PROGRAM MBUS_WZaehler (* hier wird die Klemme, an welche der M-Bus mit den Zählern angeschlossen ist, alle 10ms aufgerufen *)
VAR
	Komm_Klemme_WZaehler		: FB_MBUSKL6781;
	WMZ331_Brennwerttherme				: FB_MBUS_General_Ext;	(*1*)
	WMZ321_BHKW_1						: FB_MBUS_General_Ext;	(*3*)
	WMZ322_BHKW_2						: FB_MBUS_General_Ext;	(*4*)
	WMZ251_Druckluftkompressor			: FB_MBUS_General_Ext;	(*5*)
	WMZ215_PWT_1						: FB_MBUS_General_Ext;	(*6*)
	WMZ261_Ofenkuehlung_Dichtungen		: FB_MBUS_General_Ext;	(*7*)
	WMZ361_Abwaerme_Ofen_Abgasfackel	: FB_MBUS_General_Ext;	(*8*)
	adrBrennwerttherme				: ST_MBus_SecAdr := (udiIdNumber:=16#00474907);
	adrBHKW_1						: ST_MBus_SecAdr := (udiIdNumber:=16#00470996);
	adrBHKW_2						: ST_MBus_SecAdr := (udiIdNumber:=16#00474904);
	adrDruckluftkompressor			: ST_MBus_SecAdr := (udiIdNumber:=16#00552639);
	adrPWT_1						: ST_MBus_SecAdr := (udiIdNumber:=16#00455395);
	adrOfenkuehlung_Dichtungen		: ST_MBus_SecAdr := (udiIdNumber:=16#00482160);
	adrAbwaerme_Ofen_Abgasfackel	: ST_MBus_SecAdr := (udiIdNumber:=16#00482192);

	fbcatch : 	Error_Catch;
	fbcatch2 : 	Error_Catch;
END_VAR

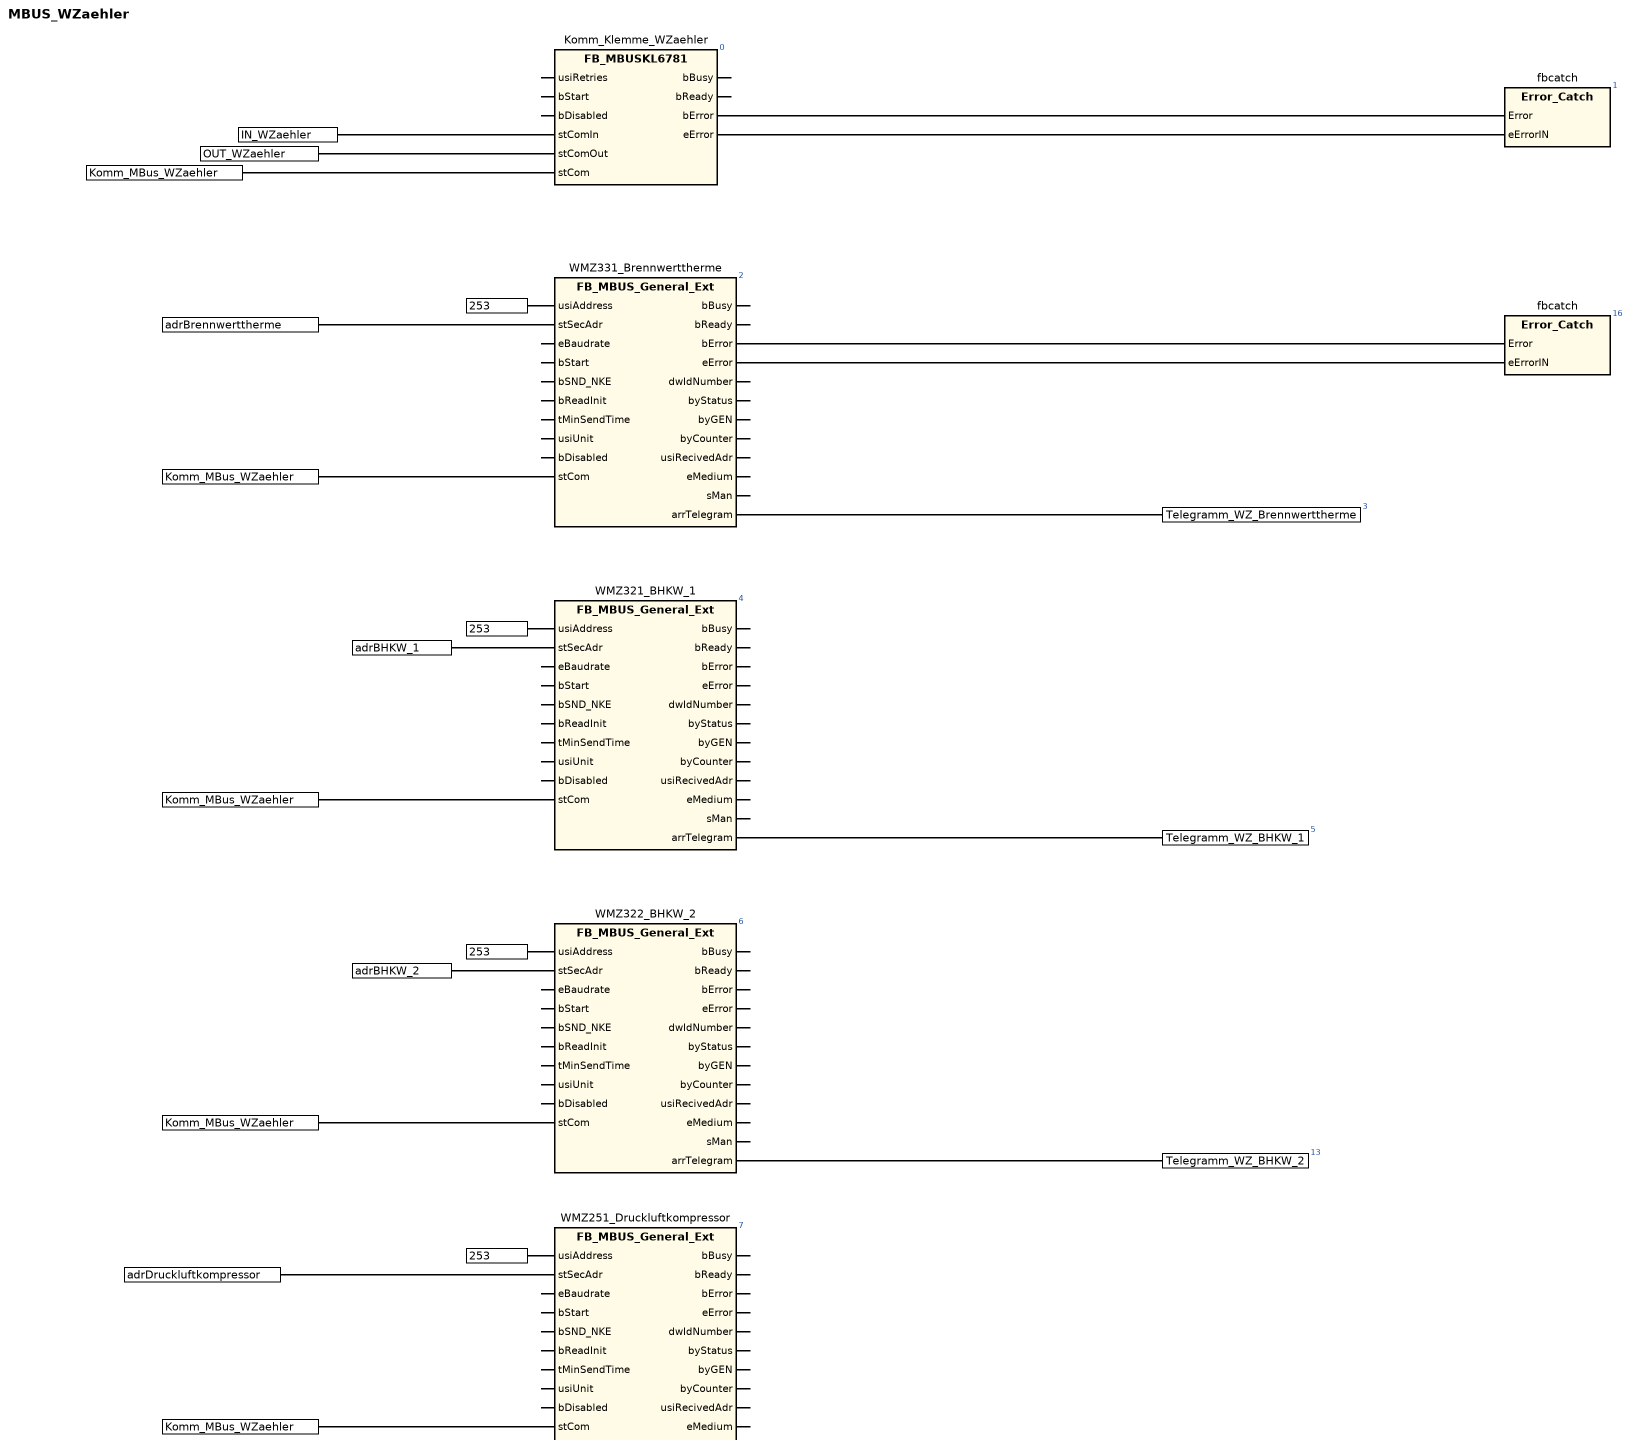
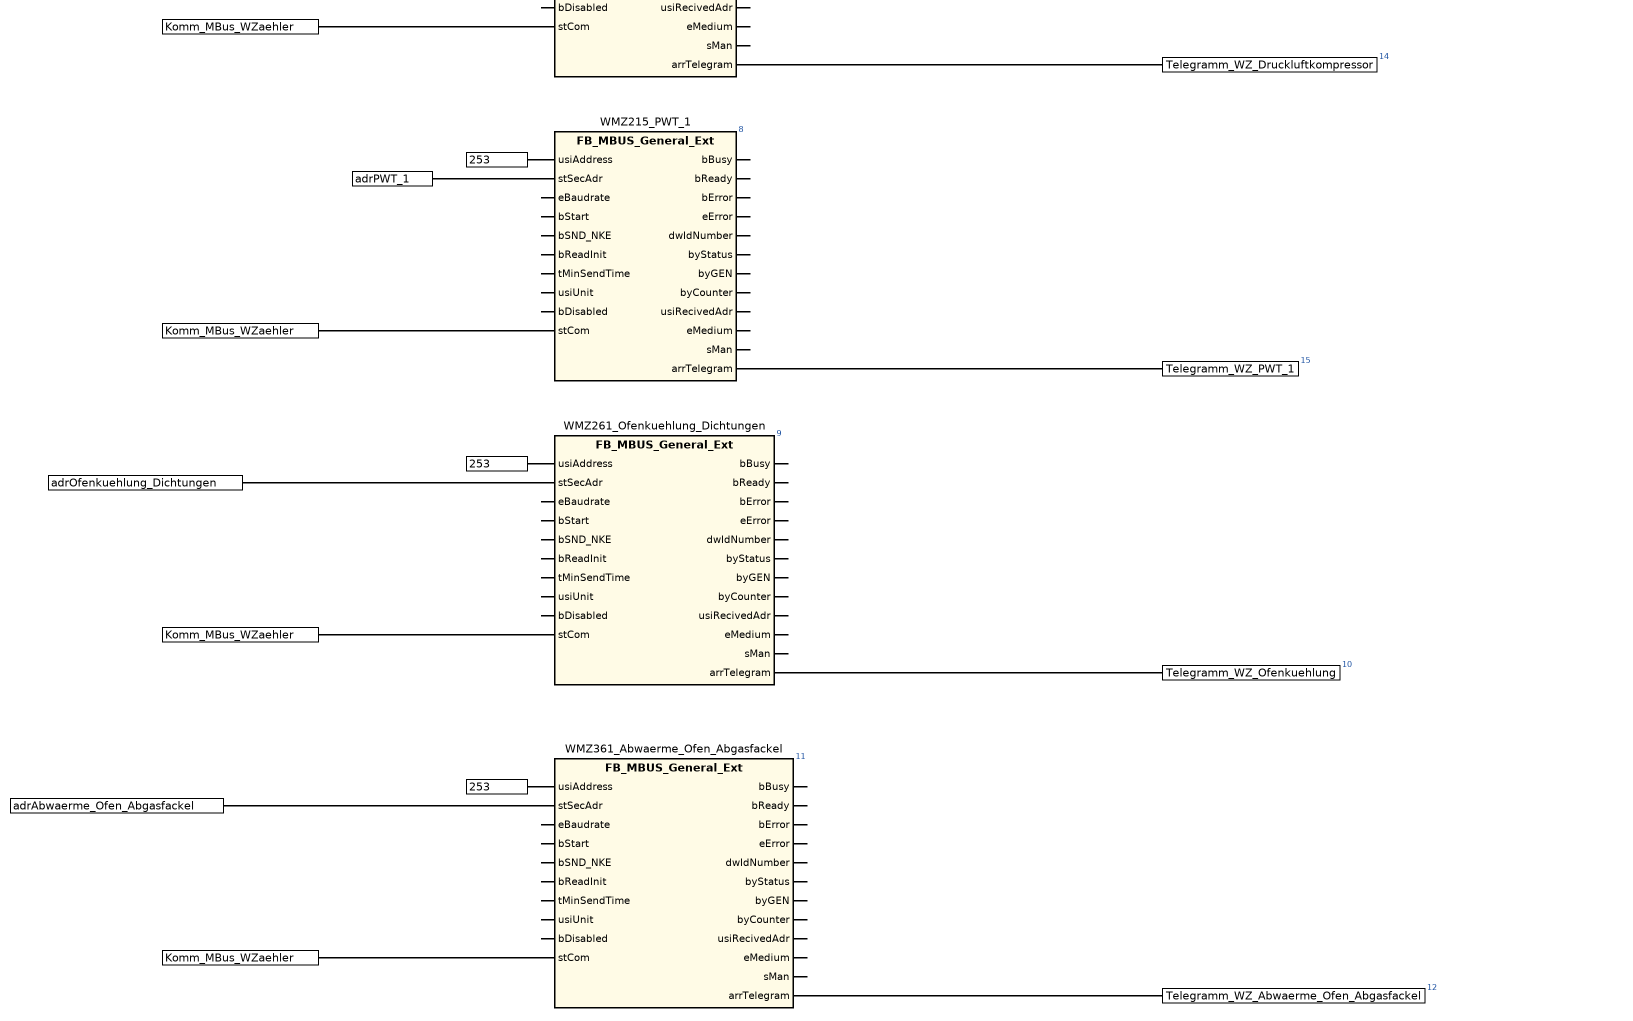
Komm_Klemme_WZaehler(stComIn := IN_WZaehler, stComOut := OUT_WZaehler, stCom := Komm_MBus_WZaehler); // FB_MBUSKL6781
fbcatch(Error := Komm_Klemme_WZaehler.bError, eErrorIN := Komm_Klemme_WZaehler.eError); // Error_Catch
WMZ331_Brennwerttherme(usiAddress := 253, stSecAdr := adrBrennwerttherme, stCom := Komm_MBus_WZaehler); // FB_MBUS_General_Ext
Telegramm_WZ_Brennwerttherme := WMZ331_Brennwerttherme.arrTelegram;
WMZ321_BHKW_1(usiAddress := 253, stSecAdr := adrBHKW_1, stCom := Komm_MBus_WZaehler); // FB_MBUS_General_Ext
Telegramm_WZ_BHKW_1 := WMZ321_BHKW_1.arrTelegram;
WMZ322_BHKW_2(usiAddress := 253, stSecAdr := adrBHKW_2, stCom := Komm_MBus_WZaehler); // FB_MBUS_General_Ext
WMZ251_Druckluftkompressor(
    usiAddress := 253,
    stSecAdr := adrDruckluftkompressor,
    stCom := Komm_MBus_WZaehler); // FB_MBUS_General_Ext
WMZ215_PWT_1(usiAddress := 253, stSecAdr := adrPWT_1, stCom := Komm_MBus_WZaehler); // FB_MBUS_General_Ext
WMZ261_Ofenkuehlung_Dichtungen(
    usiAddress := 253,
    stSecAdr := adrOfenkuehlung_Dichtungen,
    stCom := Komm_MBus_WZaehler); // FB_MBUS_General_Ext
Telegramm_WZ_Ofenkuehlung := WMZ261_Ofenkuehlung_Dichtungen.arrTelegram;
WMZ361_Abwaerme_Ofen_Abgasfackel(
    usiAddress := 253,
    stSecAdr := adrAbwaerme_Ofen_Abgasfackel,
    stCom := Komm_MBus_WZaehler); // FB_MBUS_General_Ext
Telegramm_WZ_Abwaerme_Ofen_Abgasfackel := WMZ361_Abwaerme_Ofen_Abgasfackel.arrTelegram;
Telegramm_WZ_BHKW_2 := WMZ322_BHKW_2.arrTelegram;
Telegramm_WZ_Druckluftkompressor := WMZ251_Druckluftkompressor.arrTelegram;
Telegramm_WZ_PWT_1 := WMZ215_PWT_1.arrTelegram;
fbcatch(Error := WMZ331_Brennwerttherme.bError, eErrorIN := WMZ331_Brennwerttherme.eError); // Error_Catch

END_PROGRAM

(* stored: Version 1.1.0.1, ProductVersion 3.1.4024.9
   POU MBUS_WZaehler: Id {378c9e87-39a3-460c-bc3d-585d521fd014}, SpecialFunc None *)
